PROGRAM Backbone
VAR
	RTC_FB					: RTC;
	NT_GetTime_FB			: NT_GetTime;
	RTCManagement_FB		: RTCManagement;
	FB_GetLocalAmsNetId_LU	: fb_GetLocalAmsNetId;
	bAborted				: BOOL;
	Blink_Abort				: BLINK;
	bError					: BOOL;
	Blink_Error				: BLINK;
	
	//Recipe Line 1
	Recipe_1				: FB_Recipe;
	CustomPattern_1			: RobotCustomPattern;
	Layer_1					: FB_Layer;
	
	//Recipe Line 2
	Recipe_2				: FB_Recipe;
	CustomPattern_2			: RobotCustomPattern;
	Layer_2					: FB_Layer;
	
	//Recipe Line 3
	Recipe_3				: FB_Recipe;
	CustomPattern_3			: RobotCustomPattern;
	Layer_3					: FB_Layer;
	
	//Recipe Line 4
	Recipe_4				: FB_Recipe;
	CustomPattern_4			: RobotCustomPattern;
	Layer_4					: FB_Layer;
	
	//Data Collect
	DataCollect_Palletizing_1: FGHS_DataCollect_Palletizing;
	DataCollect_Palletizing_2: FGHS_DataCollect_Palletizing;
	DataCollect_Palletizing_3: FGHS_DataCollect_Palletizing;
	DataCollect_Palletizing_4: FGHS_DataCollect_Palletizing;
	
	CheckCounter			: ARRAY [1..4] OF USINT;
	Index					: ARRAY [1..4] OF INT;
	RotatePicking			: RotatePick;
	AlarmEventHistory		: ARRAY[1..100] OF Alarm_Event_History;
	AlarmEventActive		: ARRAY[1..100] OF Alarm_Event_Active;
	OEE_Time				: OEETime;
	OEE_Time_Outfeed		: OEETime;
	bWarning				: BOOL;
	Blink_Warning			: BLINK;
	TON_Full				: TON;
	bRequest				: BOOL;
	bReleased				: BOOL;
	CheckShuttle			: FB_CheckShuttlePos;
	Check_Door				: TON;
	String_Time				: STRING(255);
	OEE_Counter				: ARRAY [1..4] OF OEECounter;
END_VAR
VAR // added by the converter: edge detectors and wires of the graphical bodies
    _w1 : BOOL;
    _rt1 : R_TRIG;
END_VAR

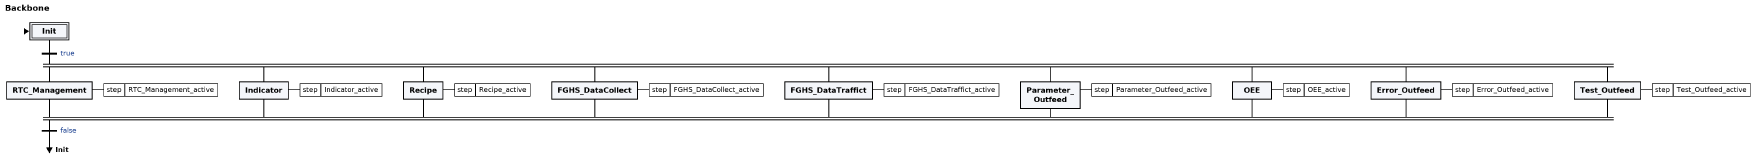
INITIAL_STEP Init:
END_STEP
TRANSITION FROM Init TO (RTC_Management, Indicator, Recipe, FGHS_DataCollect, FGHS_DataTraffict, Parameter_Outfeed, OEE, Error_Outfeed, Test_Outfeed)
    := true;
END_TRANSITION
STEP RTC_Management:
    RTC_Management_active(N);  // step action
END_STEP
STEP Indicator:
    Indicator_active(N);  // step action
END_STEP
STEP Recipe:
    Recipe_active(N);  // step action
END_STEP
STEP FGHS_DataCollect:
    FGHS_DataCollect_active(N);  // step action
END_STEP
STEP FGHS_DataTraffict:
    FGHS_DataTraffict_active(N);  // step action
END_STEP
STEP Parameter_Outfeed:
    Parameter_Outfeed_active(N);  // step action
END_STEP
STEP OEE:
    OEE_active(N);  // step action
END_STEP
STEP Error_Outfeed:
    Error_Outfeed_active(N);  // step action
END_STEP
STEP Test_Outfeed:
    Test_Outfeed_active(N);  // step action
END_STEP
TRANSITION FROM (RTC_Management, Indicator, Recipe, FGHS_DataCollect, FGHS_DataTraffict, Parameter_Outfeed, OEE, Error_Outfeed, Test_Outfeed) TO Init
    := false;
END_TRANSITION

ACTION Error_Outfeed_active:
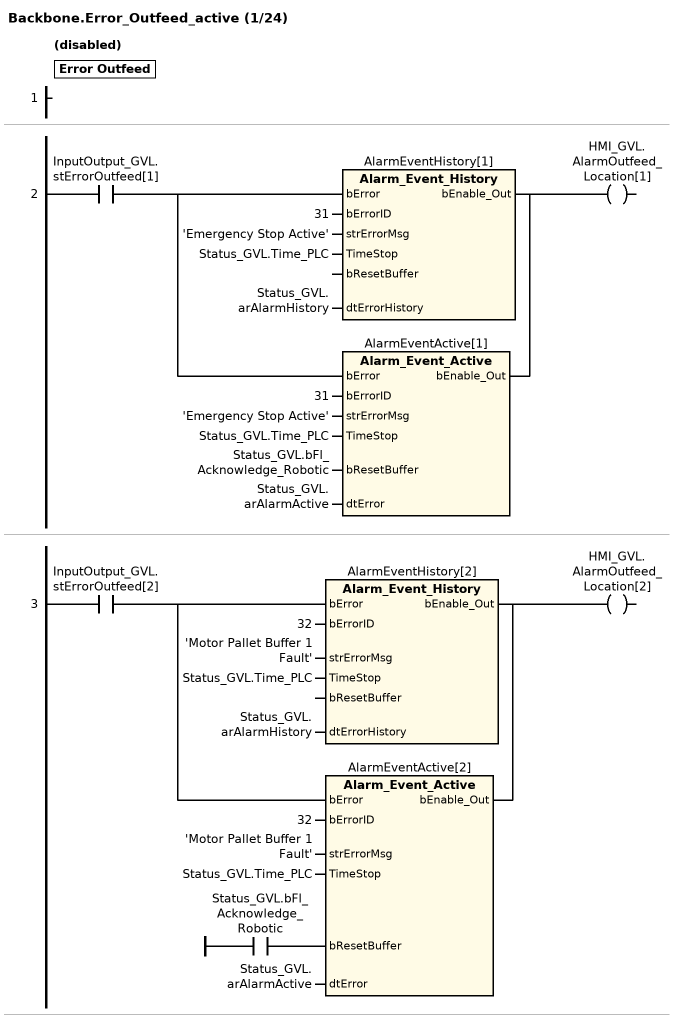
// NETWORK 1 (disabled)
// label: Error Outfeed

// NETWORK 2
AlarmEventHistory[1](
    bError := InputOutput_GVL.stErrorOutfeed[1],
    bErrorID := 31,
    strErrorMsg := 'Emergency Stop Active',
    TimeStop := Status_GVL.Time_PLC,
    dtErrorHistory := Status_GVL.arAlarmHistory); // Alarm_Event_History
AlarmEventActive[1](
    bError := InputOutput_GVL.stErrorOutfeed[1],
    bErrorID := 31,
    strErrorMsg := 'Emergency Stop Active',
    TimeStop := Status_GVL.Time_PLC,
    bResetBuffer := Status_GVL.bFl_Acknowledge_Robotic,
    dtError := Status_GVL.arAlarmActive); // Alarm_Event_Active
HMI_GVL.AlarmOutfeed_Location[1] := AlarmEventHistory[1].bEnable_Out OR AlarmEventActive[1].bEnable_Out;

// NETWORK 3
AlarmEventHistory[2](
    bError := InputOutput_GVL.stErrorOutfeed[2],
    bErrorID := 32,
    strErrorMsg := 'Motor Pallet Buffer 1 Fault',
    TimeStop := Status_GVL.Time_PLC,
    dtErrorHistory := Status_GVL.arAlarmHistory); // Alarm_Event_History
AlarmEventActive[2](
    bError := InputOutput_GVL.stErrorOutfeed[2],
    bErrorID := 32,
    strErrorMsg := 'Motor Pallet Buffer 1 Fault',
    TimeStop := Status_GVL.Time_PLC,
    bResetBuffer := Status_GVL.bFl_Acknowledge_Robotic,
    dtError := Status_GVL.arAlarmActive); // Alarm_Event_Active
HMI_GVL.AlarmOutfeed_Location[2] := AlarmEventHistory[2].bEnable_Out OR AlarmEventActive[2].bEnable_Out;

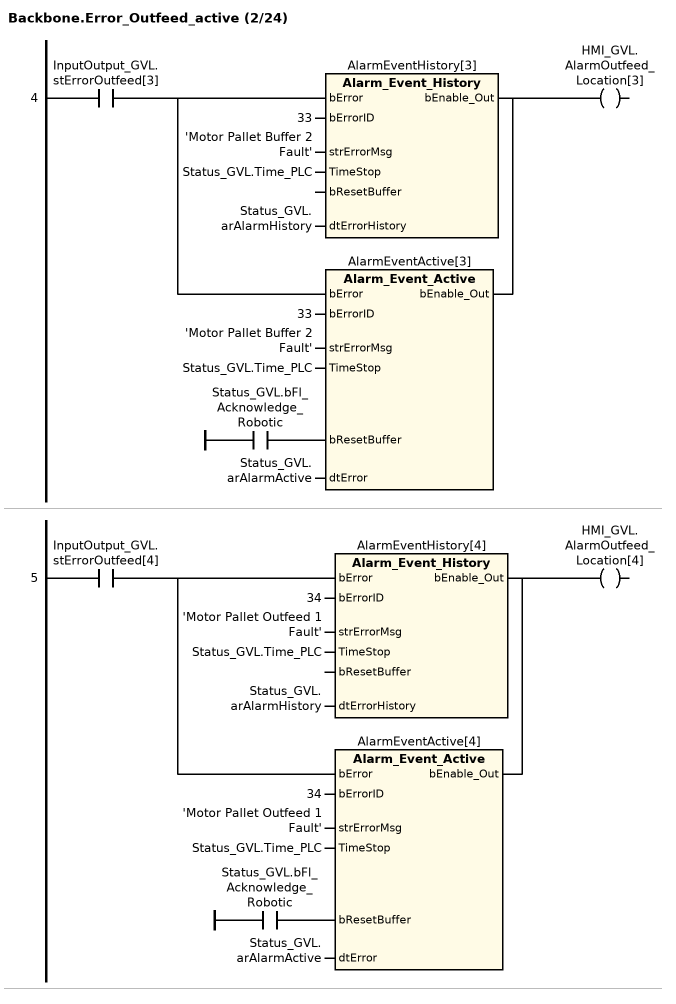
// NETWORK 4
AlarmEventHistory[3](
    bError := InputOutput_GVL.stErrorOutfeed[3],
    bErrorID := 33,
    strErrorMsg := 'Motor Pallet Buffer 2 Fault',
    TimeStop := Status_GVL.Time_PLC,
    dtErrorHistory := Status_GVL.arAlarmHistory); // Alarm_Event_History
AlarmEventActive[3](
    bError := InputOutput_GVL.stErrorOutfeed[3],
    bErrorID := 33,
    strErrorMsg := 'Motor Pallet Buffer 2 Fault',
    TimeStop := Status_GVL.Time_PLC,
    bResetBuffer := Status_GVL.bFl_Acknowledge_Robotic,
    dtError := Status_GVL.arAlarmActive); // Alarm_Event_Active
HMI_GVL.AlarmOutfeed_Location[3] := AlarmEventHistory[3].bEnable_Out OR AlarmEventActive[3].bEnable_Out;

// NETWORK 5
AlarmEventHistory[4](
    bError := InputOutput_GVL.stErrorOutfeed[4],
    bErrorID := 34,
    strErrorMsg := 'Motor Pallet Outfeed 1 Fault',
    TimeStop := Status_GVL.Time_PLC,
    dtErrorHistory := Status_GVL.arAlarmHistory); // Alarm_Event_History
AlarmEventActive[4](
    bError := InputOutput_GVL.stErrorOutfeed[4],
    bErrorID := 34,
    strErrorMsg := 'Motor Pallet Outfeed 1 Fault',
    TimeStop := Status_GVL.Time_PLC,
    bResetBuffer := Status_GVL.bFl_Acknowledge_Robotic,
    dtError := Status_GVL.arAlarmActive); // Alarm_Event_Active
HMI_GVL.AlarmOutfeed_Location[4] := AlarmEventHistory[4].bEnable_Out OR AlarmEventActive[4].bEnable_Out;

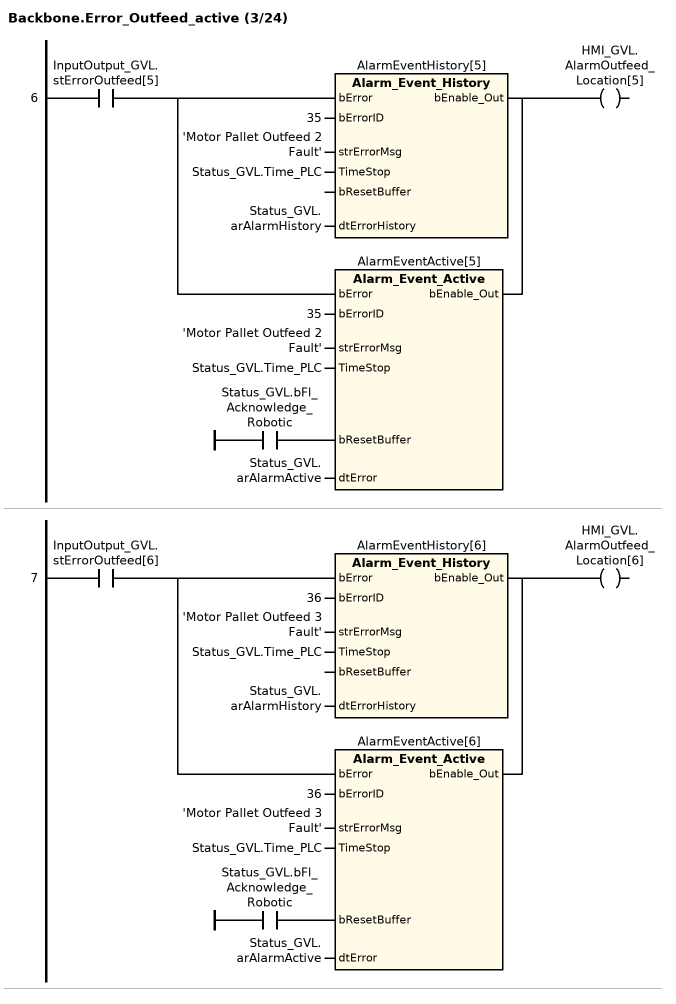
// NETWORK 6
AlarmEventHistory[5](
    bError := InputOutput_GVL.stErrorOutfeed[5],
    bErrorID := 35,
    strErrorMsg := 'Motor Pallet Outfeed 2 Fault',
    TimeStop := Status_GVL.Time_PLC,
    dtErrorHistory := Status_GVL.arAlarmHistory); // Alarm_Event_History
AlarmEventActive[5](
    bError := InputOutput_GVL.stErrorOutfeed[5],
    bErrorID := 35,
    strErrorMsg := 'Motor Pallet Outfeed 2 Fault',
    TimeStop := Status_GVL.Time_PLC,
    bResetBuffer := Status_GVL.bFl_Acknowledge_Robotic,
    dtError := Status_GVL.arAlarmActive); // Alarm_Event_Active
HMI_GVL.AlarmOutfeed_Location[5] := AlarmEventHistory[5].bEnable_Out OR AlarmEventActive[5].bEnable_Out;

// NETWORK 7
AlarmEventHistory[6](
    bError := InputOutput_GVL.stErrorOutfeed[6],
    bErrorID := 36,
    strErrorMsg := 'Motor Pallet Outfeed 3 Fault',
    TimeStop := Status_GVL.Time_PLC,
    dtErrorHistory := Status_GVL.arAlarmHistory); // Alarm_Event_History
AlarmEventActive[6](
    bError := InputOutput_GVL.stErrorOutfeed[6],
    bErrorID := 36,
    strErrorMsg := 'Motor Pallet Outfeed 3 Fault',
    TimeStop := Status_GVL.Time_PLC,
    bResetBuffer := Status_GVL.bFl_Acknowledge_Robotic,
    dtError := Status_GVL.arAlarmActive); // Alarm_Event_Active
HMI_GVL.AlarmOutfeed_Location[6] := AlarmEventHistory[6].bEnable_Out OR AlarmEventActive[6].bEnable_Out;

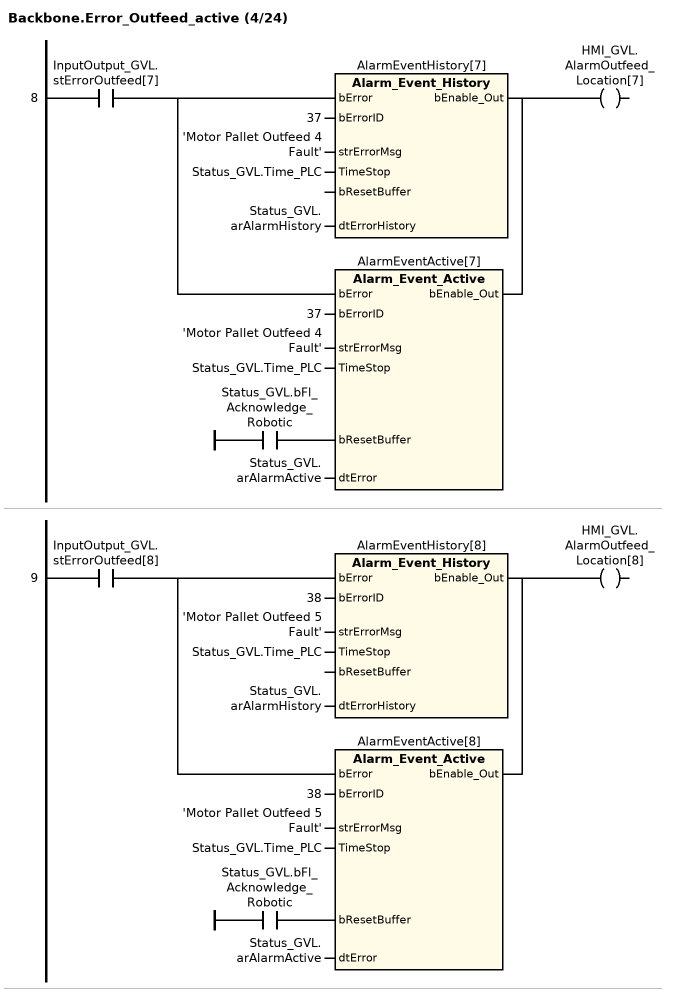
// NETWORK 8
AlarmEventHistory[7](
    bError := InputOutput_GVL.stErrorOutfeed[7],
    bErrorID := 37,
    strErrorMsg := 'Motor Pallet Outfeed 4 Fault',
    TimeStop := Status_GVL.Time_PLC,
    dtErrorHistory := Status_GVL.arAlarmHistory); // Alarm_Event_History
AlarmEventActive[7](
    bError := InputOutput_GVL.stErrorOutfeed[7],
    bErrorID := 37,
    strErrorMsg := 'Motor Pallet Outfeed 4 Fault',
    TimeStop := Status_GVL.Time_PLC,
    bResetBuffer := Status_GVL.bFl_Acknowledge_Robotic,
    dtError := Status_GVL.arAlarmActive); // Alarm_Event_Active
HMI_GVL.AlarmOutfeed_Location[7] := AlarmEventHistory[7].bEnable_Out OR AlarmEventActive[7].bEnable_Out;

// NETWORK 9
AlarmEventHistory[8](
    bError := InputOutput_GVL.stErrorOutfeed[8],
    bErrorID := 38,
    strErrorMsg := 'Motor Pallet Outfeed 5 Fault',
    TimeStop := Status_GVL.Time_PLC,
    dtErrorHistory := Status_GVL.arAlarmHistory); // Alarm_Event_History
AlarmEventActive[8](
    bError := InputOutput_GVL.stErrorOutfeed[8],
    bErrorID := 38,
    strErrorMsg := 'Motor Pallet Outfeed 5 Fault',
    TimeStop := Status_GVL.Time_PLC,
    bResetBuffer := Status_GVL.bFl_Acknowledge_Robotic,
    dtError := Status_GVL.arAlarmActive); // Alarm_Event_Active
HMI_GVL.AlarmOutfeed_Location[8] := AlarmEventHistory[8].bEnable_Out OR AlarmEventActive[8].bEnable_Out;

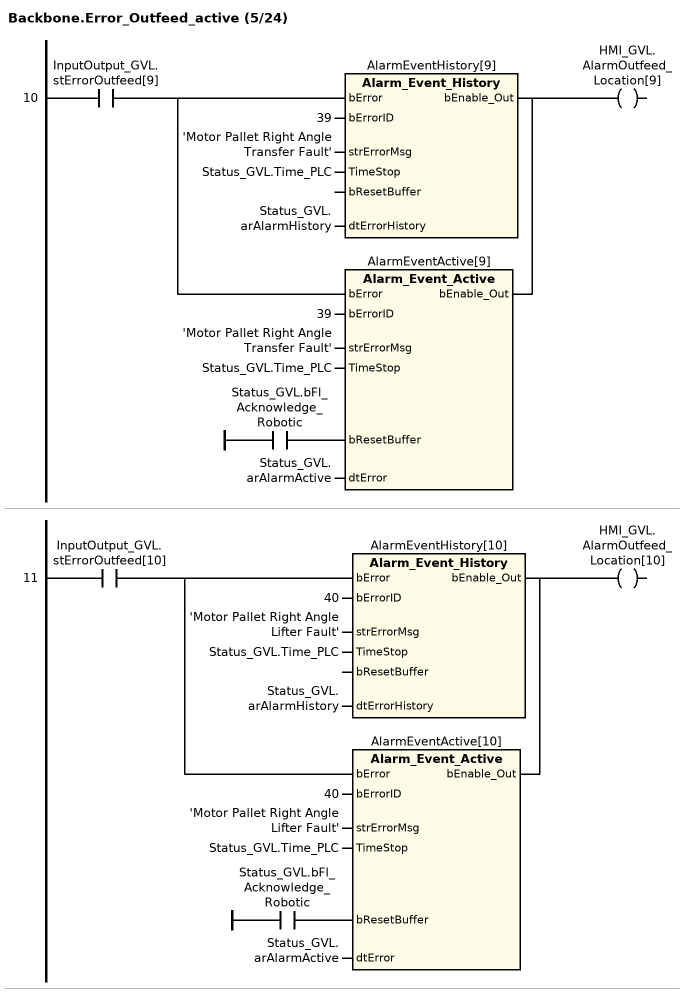
// NETWORK 10
AlarmEventHistory[9](
    bError := InputOutput_GVL.stErrorOutfeed[9],
    bErrorID := 39,
    strErrorMsg := 'Motor Pallet Right Angle Transfer Fault',
    TimeStop := Status_GVL.Time_PLC,
    dtErrorHistory := Status_GVL.arAlarmHistory); // Alarm_Event_History
AlarmEventActive[9](
    bError := InputOutput_GVL.stErrorOutfeed[9],
    bErrorID := 39,
    strErrorMsg := 'Motor Pallet Right Angle Transfer Fault',
    TimeStop := Status_GVL.Time_PLC,
    bResetBuffer := Status_GVL.bFl_Acknowledge_Robotic,
    dtError := Status_GVL.arAlarmActive); // Alarm_Event_Active
HMI_GVL.AlarmOutfeed_Location[9] := AlarmEventHistory[9].bEnable_Out OR AlarmEventActive[9].bEnable_Out;

// NETWORK 11
AlarmEventHistory[10](
    bError := InputOutput_GVL.stErrorOutfeed[10],
    bErrorID := 40,
    strErrorMsg := 'Motor Pallet Right Angle Lifter Fault',
    TimeStop := Status_GVL.Time_PLC,
    dtErrorHistory := Status_GVL.arAlarmHistory); // Alarm_Event_History
AlarmEventActive[10](
    bError := InputOutput_GVL.stErrorOutfeed[10],
    bErrorID := 40,
    strErrorMsg := 'Motor Pallet Right Angle Lifter Fault',
    TimeStop := Status_GVL.Time_PLC,
    bResetBuffer := Status_GVL.bFl_Acknowledge_Robotic,
    dtError := Status_GVL.arAlarmActive); // Alarm_Event_Active
HMI_GVL.AlarmOutfeed_Location[10] := AlarmEventHistory[10].bEnable_Out OR AlarmEventActive[10].bEnable_Out;

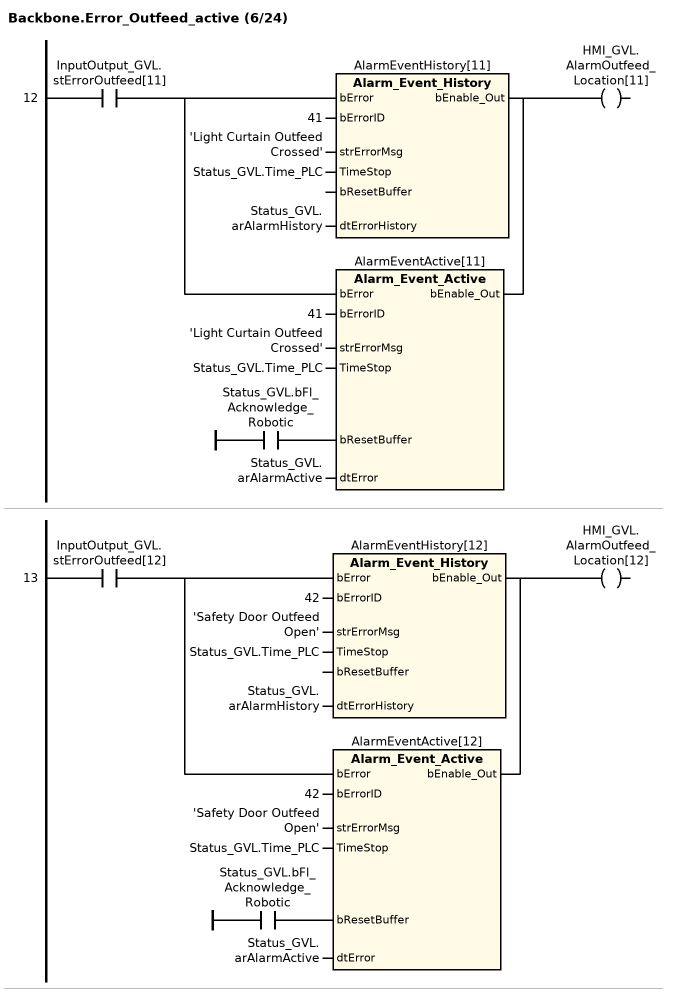
// NETWORK 12
AlarmEventHistory[11](
    bError := InputOutput_GVL.stErrorOutfeed[11],
    bErrorID := 41,
    strErrorMsg := 'Light Curtain Outfeed Crossed',
    TimeStop := Status_GVL.Time_PLC,
    dtErrorHistory := Status_GVL.arAlarmHistory); // Alarm_Event_History
AlarmEventActive[11](
    bError := InputOutput_GVL.stErrorOutfeed[11],
    bErrorID := 41,
    strErrorMsg := 'Light Curtain Outfeed Crossed',
    TimeStop := Status_GVL.Time_PLC,
    bResetBuffer := Status_GVL.bFl_Acknowledge_Robotic,
    dtError := Status_GVL.arAlarmActive); // Alarm_Event_Active
HMI_GVL.AlarmOutfeed_Location[11] := AlarmEventHistory[11].bEnable_Out OR AlarmEventActive[11].bEnable_Out;

// NETWORK 13
AlarmEventHistory[12](
    bError := InputOutput_GVL.stErrorOutfeed[12],
    bErrorID := 42,
    strErrorMsg := 'Safety Door Outfeed Open',
    TimeStop := Status_GVL.Time_PLC,
    dtErrorHistory := Status_GVL.arAlarmHistory); // Alarm_Event_History
AlarmEventActive[12](
    bError := InputOutput_GVL.stErrorOutfeed[12],
    bErrorID := 42,
    strErrorMsg := 'Safety Door Outfeed Open',
    TimeStop := Status_GVL.Time_PLC,
    bResetBuffer := Status_GVL.bFl_Acknowledge_Robotic,
    dtError := Status_GVL.arAlarmActive); // Alarm_Event_Active
HMI_GVL.AlarmOutfeed_Location[12] := AlarmEventHistory[12].bEnable_Out OR AlarmEventActive[12].bEnable_Out;

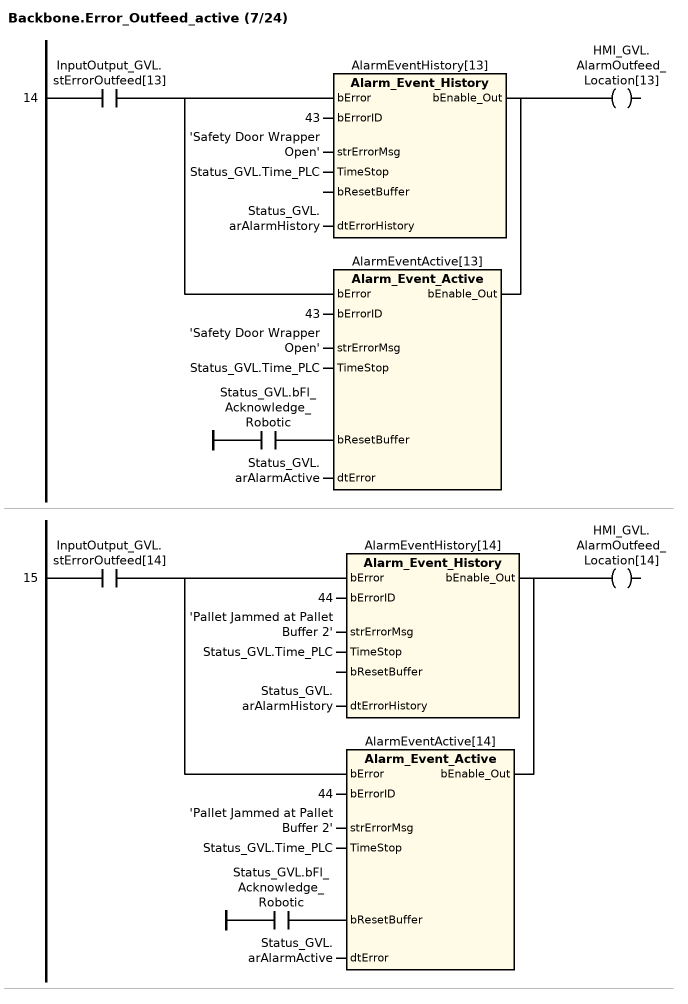
// NETWORK 14
AlarmEventHistory[13](
    bError := InputOutput_GVL.stErrorOutfeed[13],
    bErrorID := 43,
    strErrorMsg := 'Safety Door Wrapper Open',
    TimeStop := Status_GVL.Time_PLC,
    dtErrorHistory := Status_GVL.arAlarmHistory); // Alarm_Event_History
AlarmEventActive[13](
    bError := InputOutput_GVL.stErrorOutfeed[13],
    bErrorID := 43,
    strErrorMsg := 'Safety Door Wrapper Open',
    TimeStop := Status_GVL.Time_PLC,
    bResetBuffer := Status_GVL.bFl_Acknowledge_Robotic,
    dtError := Status_GVL.arAlarmActive); // Alarm_Event_Active
HMI_GVL.AlarmOutfeed_Location[13] := AlarmEventHistory[13].bEnable_Out OR AlarmEventActive[13].bEnable_Out;

// NETWORK 15
AlarmEventHistory[14](
    bError := InputOutput_GVL.stErrorOutfeed[14],
    bErrorID := 44,
    strErrorMsg := 'Pallet Jammed at Pallet Buffer 2',
    TimeStop := Status_GVL.Time_PLC,
    dtErrorHistory := Status_GVL.arAlarmHistory); // Alarm_Event_History
AlarmEventActive[14](
    bError := InputOutput_GVL.stErrorOutfeed[14],
    bErrorID := 44,
    strErrorMsg := 'Pallet Jammed at Pallet Buffer 2',
    TimeStop := Status_GVL.Time_PLC,
    bResetBuffer := Status_GVL.bFl_Acknowledge_Robotic,
    dtError := Status_GVL.arAlarmActive); // Alarm_Event_Active
HMI_GVL.AlarmOutfeed_Location[14] := AlarmEventHistory[14].bEnable_Out OR AlarmEventActive[14].bEnable_Out;

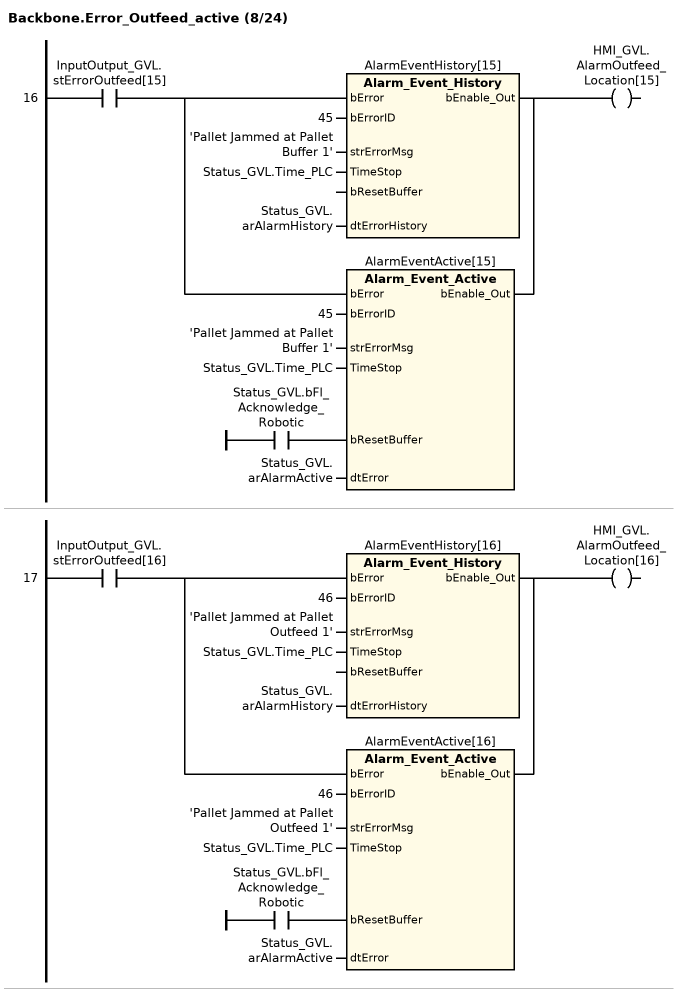
// NETWORK 16
AlarmEventHistory[15](
    bError := InputOutput_GVL.stErrorOutfeed[15],
    bErrorID := 45,
    strErrorMsg := 'Pallet Jammed at Pallet Buffer 1',
    TimeStop := Status_GVL.Time_PLC,
    dtErrorHistory := Status_GVL.arAlarmHistory); // Alarm_Event_History
AlarmEventActive[15](
    bError := InputOutput_GVL.stErrorOutfeed[15],
    bErrorID := 45,
    strErrorMsg := 'Pallet Jammed at Pallet Buffer 1',
    TimeStop := Status_GVL.Time_PLC,
    bResetBuffer := Status_GVL.bFl_Acknowledge_Robotic,
    dtError := Status_GVL.arAlarmActive); // Alarm_Event_Active
HMI_GVL.AlarmOutfeed_Location[15] := AlarmEventHistory[15].bEnable_Out OR AlarmEventActive[15].bEnable_Out;

// NETWORK 17
AlarmEventHistory[16](
    bError := InputOutput_GVL.stErrorOutfeed[16],
    bErrorID := 46,
    strErrorMsg := 'Pallet Jammed at Pallet Outfeed 1',
    TimeStop := Status_GVL.Time_PLC,
    dtErrorHistory := Status_GVL.arAlarmHistory); // Alarm_Event_History
AlarmEventActive[16](
    bError := InputOutput_GVL.stErrorOutfeed[16],
    bErrorID := 46,
    strErrorMsg := 'Pallet Jammed at Pallet Outfeed 1',
    TimeStop := Status_GVL.Time_PLC,
    bResetBuffer := Status_GVL.bFl_Acknowledge_Robotic,
    dtError := Status_GVL.arAlarmActive); // Alarm_Event_Active
HMI_GVL.AlarmOutfeed_Location[16] := AlarmEventHistory[16].bEnable_Out OR AlarmEventActive[16].bEnable_Out;

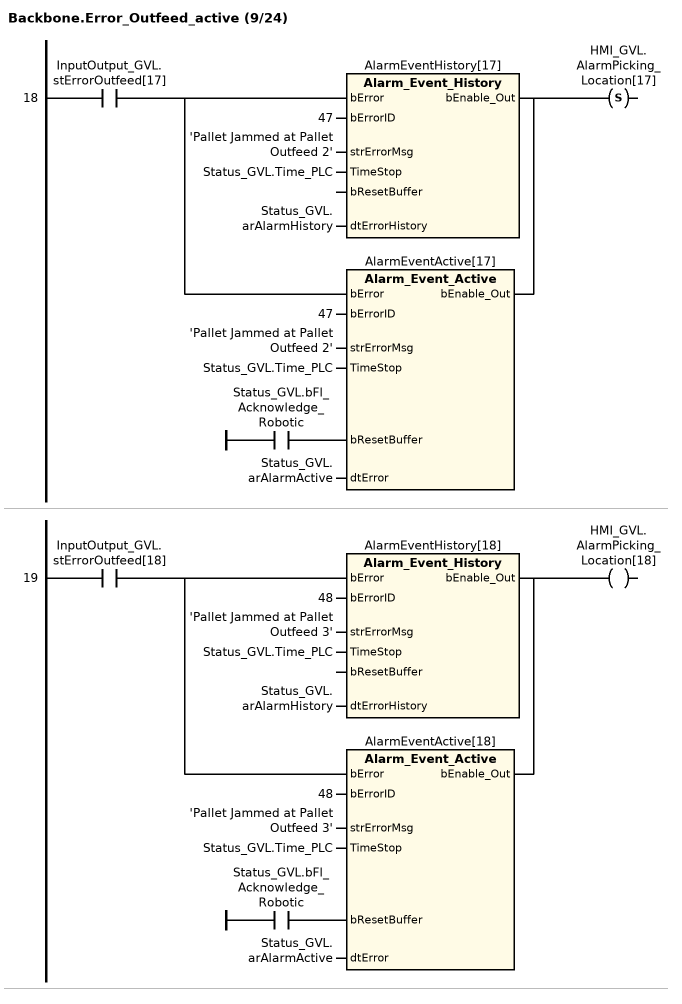
// NETWORK 18
AlarmEventHistory[17](
    bError := InputOutput_GVL.stErrorOutfeed[17],
    bErrorID := 47,
    strErrorMsg := 'Pallet Jammed at Pallet Outfeed 2',
    TimeStop := Status_GVL.Time_PLC,
    dtErrorHistory := Status_GVL.arAlarmHistory); // Alarm_Event_History
AlarmEventActive[17](
    bError := InputOutput_GVL.stErrorOutfeed[17],
    bErrorID := 47,
    strErrorMsg := 'Pallet Jammed at Pallet Outfeed 2',
    TimeStop := Status_GVL.Time_PLC,
    bResetBuffer := Status_GVL.bFl_Acknowledge_Robotic,
    dtError := Status_GVL.arAlarmActive); // Alarm_Event_Active
HMI_GVL.AlarmPicking_Location[17] S= AlarmEventHistory[17].bEnable_Out OR AlarmEventActive[17].bEnable_Out;

// NETWORK 19
AlarmEventHistory[18](
    bError := InputOutput_GVL.stErrorOutfeed[18],
    bErrorID := 48,
    strErrorMsg := 'Pallet Jammed at Pallet Outfeed 3',
    TimeStop := Status_GVL.Time_PLC,
    dtErrorHistory := Status_GVL.arAlarmHistory); // Alarm_Event_History
AlarmEventActive[18](
    bError := InputOutput_GVL.stErrorOutfeed[18],
    bErrorID := 48,
    strErrorMsg := 'Pallet Jammed at Pallet Outfeed 3',
    TimeStop := Status_GVL.Time_PLC,
    bResetBuffer := Status_GVL.bFl_Acknowledge_Robotic,
    dtError := Status_GVL.arAlarmActive); // Alarm_Event_Active
HMI_GVL.AlarmPicking_Location[18] := AlarmEventHistory[18].bEnable_Out OR AlarmEventActive[18].bEnable_Out;

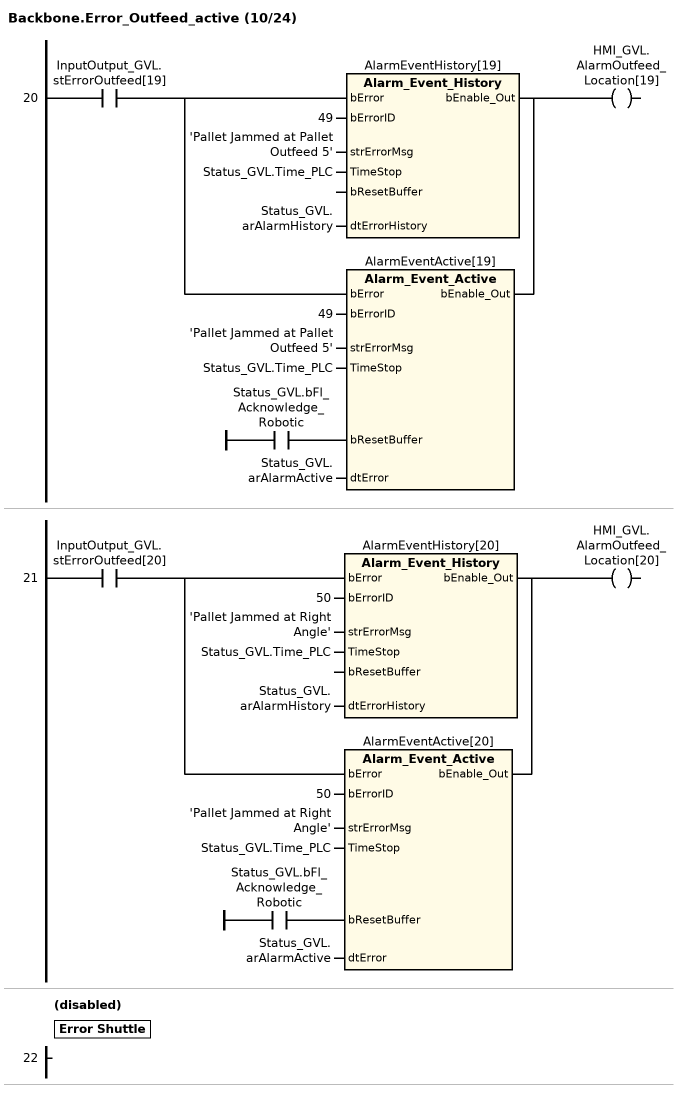
// NETWORK 20
AlarmEventHistory[19](
    bError := InputOutput_GVL.stErrorOutfeed[19],
    bErrorID := 49,
    strErrorMsg := 'Pallet Jammed at Pallet Outfeed 5',
    TimeStop := Status_GVL.Time_PLC,
    dtErrorHistory := Status_GVL.arAlarmHistory); // Alarm_Event_History
AlarmEventActive[19](
    bError := InputOutput_GVL.stErrorOutfeed[19],
    bErrorID := 49,
    strErrorMsg := 'Pallet Jammed at Pallet Outfeed 5',
    TimeStop := Status_GVL.Time_PLC,
    bResetBuffer := Status_GVL.bFl_Acknowledge_Robotic,
    dtError := Status_GVL.arAlarmActive); // Alarm_Event_Active
HMI_GVL.AlarmOutfeed_Location[19] := AlarmEventHistory[19].bEnable_Out OR AlarmEventActive[19].bEnable_Out;

// NETWORK 21
AlarmEventHistory[20](
    bError := InputOutput_GVL.stErrorOutfeed[20],
    bErrorID := 50,
    strErrorMsg := 'Pallet Jammed at Right Angle',
    TimeStop := Status_GVL.Time_PLC,
    dtErrorHistory := Status_GVL.arAlarmHistory); // Alarm_Event_History
AlarmEventActive[20](
    bError := InputOutput_GVL.stErrorOutfeed[20],
    bErrorID := 50,
    strErrorMsg := 'Pallet Jammed at Right Angle',
    TimeStop := Status_GVL.Time_PLC,
    bResetBuffer := Status_GVL.bFl_Acknowledge_Robotic,
    dtError := Status_GVL.arAlarmActive); // Alarm_Event_Active
HMI_GVL.AlarmOutfeed_Location[20] := AlarmEventHistory[20].bEnable_Out OR AlarmEventActive[20].bEnable_Out;

// NETWORK 22 (disabled)
// label: Error Shuttle

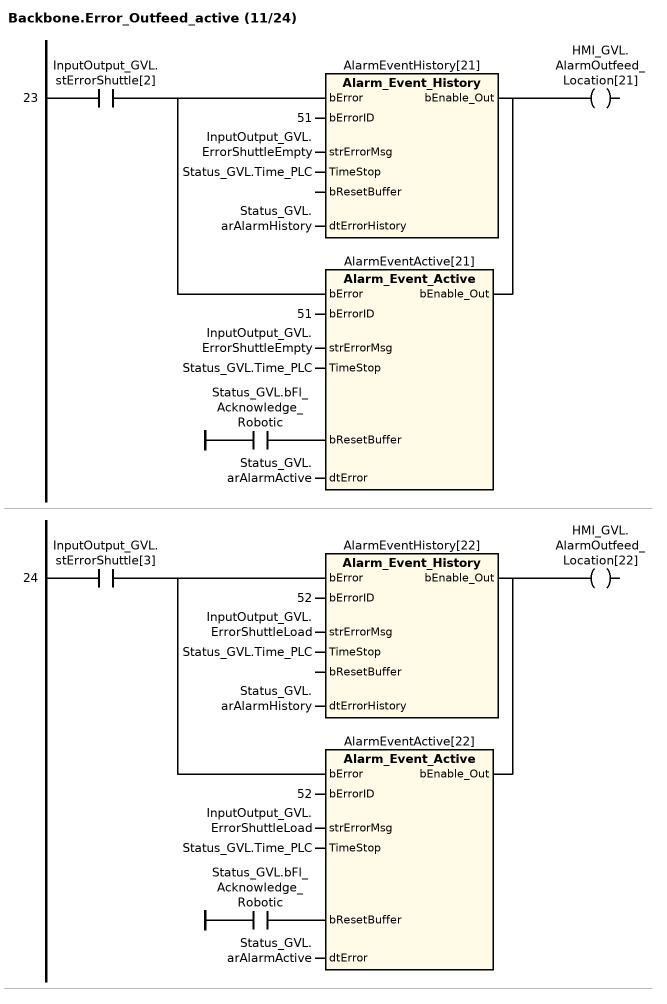
// NETWORK 23
AlarmEventHistory[21](
    bError := InputOutput_GVL.stErrorShuttle[2],
    bErrorID := 51,
    strErrorMsg := InputOutput_GVL.ErrorShuttleEmpty,
    TimeStop := Status_GVL.Time_PLC,
    dtErrorHistory := Status_GVL.arAlarmHistory); // Alarm_Event_History
AlarmEventActive[21](
    bError := InputOutput_GVL.stErrorShuttle[2],
    bErrorID := 51,
    strErrorMsg := InputOutput_GVL.ErrorShuttleEmpty,
    TimeStop := Status_GVL.Time_PLC,
    bResetBuffer := Status_GVL.bFl_Acknowledge_Robotic,
    dtError := Status_GVL.arAlarmActive); // Alarm_Event_Active
HMI_GVL.AlarmOutfeed_Location[21] := AlarmEventHistory[21].bEnable_Out OR AlarmEventActive[21].bEnable_Out;

// NETWORK 24
AlarmEventHistory[22](
    bError := InputOutput_GVL.stErrorShuttle[3],
    bErrorID := 52,
    strErrorMsg := InputOutput_GVL.ErrorShuttleLoad,
    TimeStop := Status_GVL.Time_PLC,
    dtErrorHistory := Status_GVL.arAlarmHistory); // Alarm_Event_History
AlarmEventActive[22](
    bError := InputOutput_GVL.stErrorShuttle[3],
    bErrorID := 52,
    strErrorMsg := InputOutput_GVL.ErrorShuttleLoad,
    TimeStop := Status_GVL.Time_PLC,
    bResetBuffer := Status_GVL.bFl_Acknowledge_Robotic,
    dtError := Status_GVL.arAlarmActive); // Alarm_Event_Active
HMI_GVL.AlarmOutfeed_Location[22] := AlarmEventHistory[22].bEnable_Out OR AlarmEventActive[22].bEnable_Out;

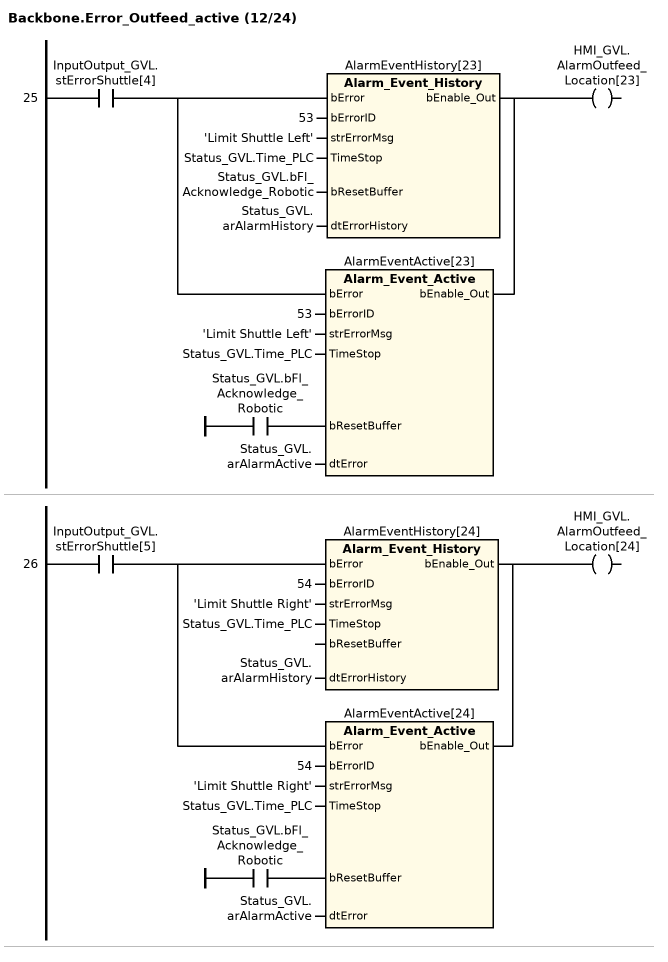
// NETWORK 25
AlarmEventHistory[23](
    bError := InputOutput_GVL.stErrorShuttle[4],
    bErrorID := 53,
    strErrorMsg := 'Limit Shuttle Left',
    TimeStop := Status_GVL.Time_PLC,
    bResetBuffer := Status_GVL.bFl_Acknowledge_Robotic,
    dtErrorHistory := Status_GVL.arAlarmHistory); // Alarm_Event_History
AlarmEventActive[23](
    bError := InputOutput_GVL.stErrorShuttle[4],
    bErrorID := 53,
    strErrorMsg := 'Limit Shuttle Left',
    TimeStop := Status_GVL.Time_PLC,
    bResetBuffer := Status_GVL.bFl_Acknowledge_Robotic,
    dtError := Status_GVL.arAlarmActive); // Alarm_Event_Active
HMI_GVL.AlarmOutfeed_Location[23] := AlarmEventHistory[23].bEnable_Out OR AlarmEventActive[23].bEnable_Out;

// NETWORK 26
AlarmEventHistory[24](
    bError := InputOutput_GVL.stErrorShuttle[5],
    bErrorID := 54,
    strErrorMsg := 'Limit Shuttle Right',
    TimeStop := Status_GVL.Time_PLC,
    dtErrorHistory := Status_GVL.arAlarmHistory); // Alarm_Event_History
AlarmEventActive[24](
    bError := InputOutput_GVL.stErrorShuttle[5],
    bErrorID := 54,
    strErrorMsg := 'Limit Shuttle Right',
    TimeStop := Status_GVL.Time_PLC,
    bResetBuffer := Status_GVL.bFl_Acknowledge_Robotic,
    dtError := Status_GVL.arAlarmActive); // Alarm_Event_Active
HMI_GVL.AlarmOutfeed_Location[24] := AlarmEventHistory[24].bEnable_Out OR AlarmEventActive[24].bEnable_Out;

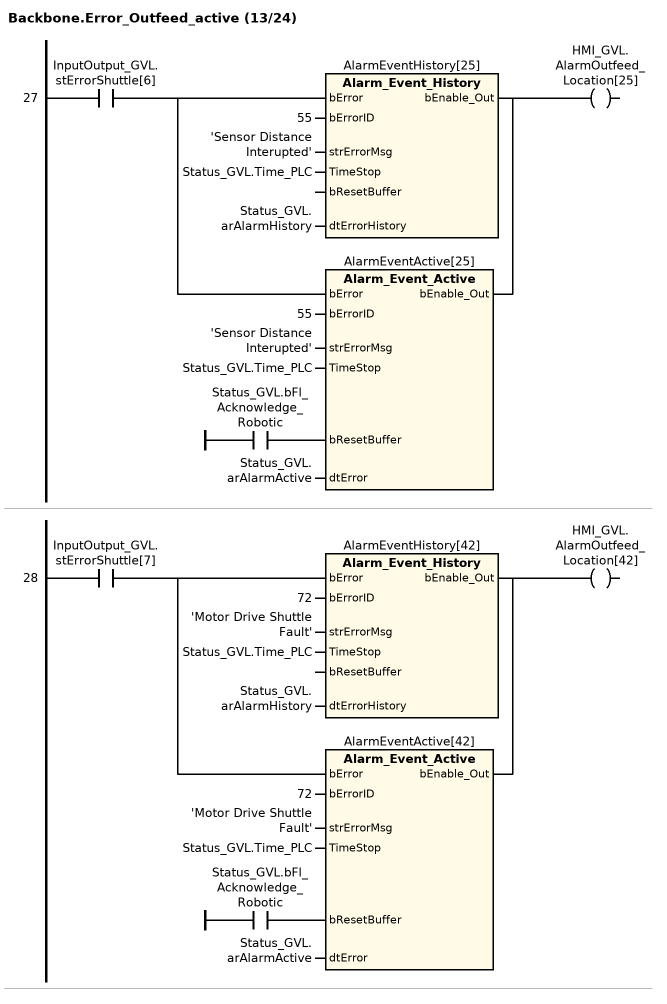
// NETWORK 27
AlarmEventHistory[25](
    bError := InputOutput_GVL.stErrorShuttle[6],
    bErrorID := 55,
    strErrorMsg := 'Sensor Distance Interupted',
    TimeStop := Status_GVL.Time_PLC,
    dtErrorHistory := Status_GVL.arAlarmHistory); // Alarm_Event_History
AlarmEventActive[25](
    bError := InputOutput_GVL.stErrorShuttle[6],
    bErrorID := 55,
    strErrorMsg := 'Sensor Distance Interupted',
    TimeStop := Status_GVL.Time_PLC,
    bResetBuffer := Status_GVL.bFl_Acknowledge_Robotic,
    dtError := Status_GVL.arAlarmActive); // Alarm_Event_Active
HMI_GVL.AlarmOutfeed_Location[25] := AlarmEventHistory[25].bEnable_Out OR AlarmEventActive[25].bEnable_Out;

// NETWORK 28
AlarmEventHistory[42](
    bError := InputOutput_GVL.stErrorShuttle[7],
    bErrorID := 72,
    strErrorMsg := 'Motor Drive Shuttle Fault',
    TimeStop := Status_GVL.Time_PLC,
    dtErrorHistory := Status_GVL.arAlarmHistory); // Alarm_Event_History
AlarmEventActive[42](
    bError := InputOutput_GVL.stErrorShuttle[7],
    bErrorID := 72,
    strErrorMsg := 'Motor Drive Shuttle Fault',
    TimeStop := Status_GVL.Time_PLC,
    bResetBuffer := Status_GVL.bFl_Acknowledge_Robotic,
    dtError := Status_GVL.arAlarmActive); // Alarm_Event_Active
HMI_GVL.AlarmOutfeed_Location[42] := AlarmEventHistory[42].bEnable_Out OR AlarmEventActive[42].bEnable_Out;

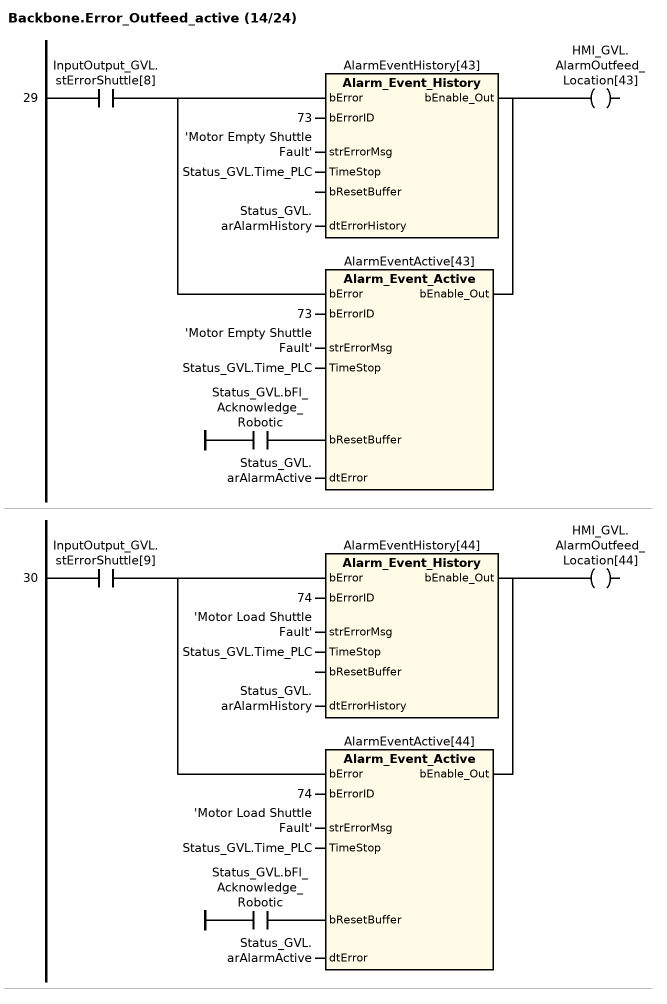
// NETWORK 29
AlarmEventHistory[43](
    bError := InputOutput_GVL.stErrorShuttle[8],
    bErrorID := 73,
    strErrorMsg := 'Motor Empty Shuttle Fault',
    TimeStop := Status_GVL.Time_PLC,
    dtErrorHistory := Status_GVL.arAlarmHistory); // Alarm_Event_History
AlarmEventActive[43](
    bError := InputOutput_GVL.stErrorShuttle[8],
    bErrorID := 73,
    strErrorMsg := 'Motor Empty Shuttle Fault',
    TimeStop := Status_GVL.Time_PLC,
    bResetBuffer := Status_GVL.bFl_Acknowledge_Robotic,
    dtError := Status_GVL.arAlarmActive); // Alarm_Event_Active
HMI_GVL.AlarmOutfeed_Location[43] := AlarmEventHistory[43].bEnable_Out OR AlarmEventActive[43].bEnable_Out;

// NETWORK 30
AlarmEventHistory[44](
    bError := InputOutput_GVL.stErrorShuttle[9],
    bErrorID := 74,
    strErrorMsg := 'Motor Load Shuttle Fault',
    TimeStop := Status_GVL.Time_PLC,
    dtErrorHistory := Status_GVL.arAlarmHistory); // Alarm_Event_History
AlarmEventActive[44](
    bError := InputOutput_GVL.stErrorShuttle[9],
    bErrorID := 74,
    strErrorMsg := 'Motor Load Shuttle Fault',
    TimeStop := Status_GVL.Time_PLC,
    bResetBuffer := Status_GVL.bFl_Acknowledge_Robotic,
    dtError := Status_GVL.arAlarmActive); // Alarm_Event_Active
HMI_GVL.AlarmOutfeed_Location[44] := AlarmEventHistory[44].bEnable_Out OR AlarmEventActive[44].bEnable_Out;

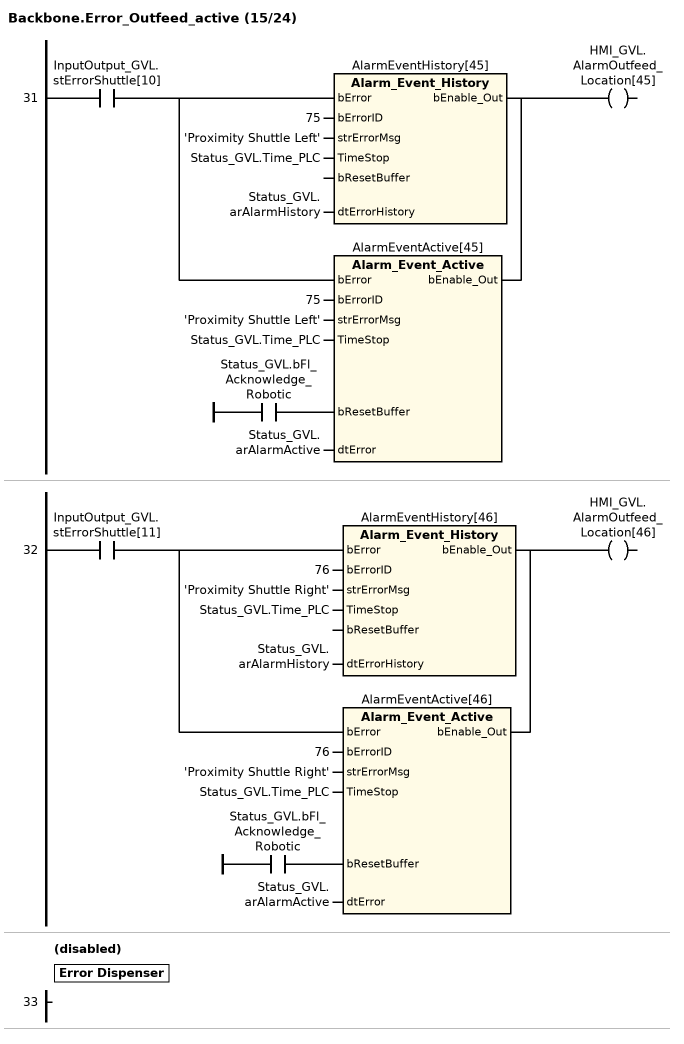
// NETWORK 31
AlarmEventHistory[45](
    bError := InputOutput_GVL.stErrorShuttle[10],
    bErrorID := 75,
    strErrorMsg := 'Proximity Shuttle Left',
    TimeStop := Status_GVL.Time_PLC,
    dtErrorHistory := Status_GVL.arAlarmHistory); // Alarm_Event_History
AlarmEventActive[45](
    bError := InputOutput_GVL.stErrorShuttle[10],
    bErrorID := 75,
    strErrorMsg := 'Proximity Shuttle Left',
    TimeStop := Status_GVL.Time_PLC,
    bResetBuffer := Status_GVL.bFl_Acknowledge_Robotic,
    dtError := Status_GVL.arAlarmActive); // Alarm_Event_Active
HMI_GVL.AlarmOutfeed_Location[45] := AlarmEventHistory[45].bEnable_Out OR AlarmEventActive[45].bEnable_Out;

// NETWORK 32
AlarmEventHistory[46](
    bError := InputOutput_GVL.stErrorShuttle[11],
    bErrorID := 76,
    strErrorMsg := 'Proximity Shuttle Right',
    TimeStop := Status_GVL.Time_PLC,
    dtErrorHistory := Status_GVL.arAlarmHistory); // Alarm_Event_History
AlarmEventActive[46](
    bError := InputOutput_GVL.stErrorShuttle[11],
    bErrorID := 76,
    strErrorMsg := 'Proximity Shuttle Right',
    TimeStop := Status_GVL.Time_PLC,
    bResetBuffer := Status_GVL.bFl_Acknowledge_Robotic,
    dtError := Status_GVL.arAlarmActive); // Alarm_Event_Active
HMI_GVL.AlarmOutfeed_Location[46] := AlarmEventHistory[46].bEnable_Out OR AlarmEventActive[46].bEnable_Out;

// NETWORK 33 (disabled)
// label: Error Dispenser

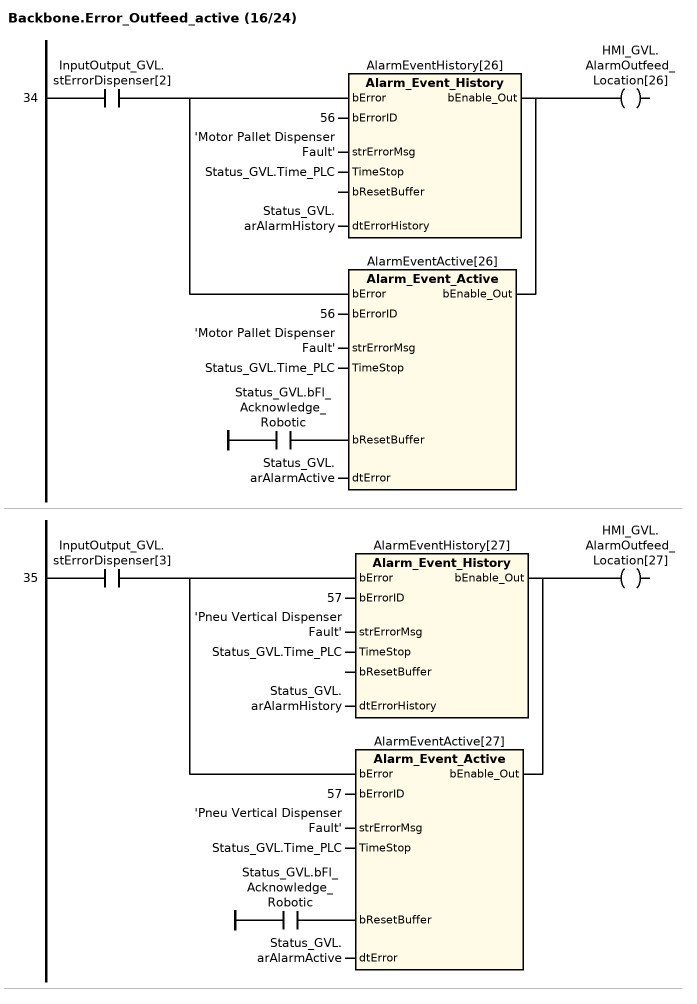
// NETWORK 34
AlarmEventHistory[26](
    bError := InputOutput_GVL.stErrorDispenser[2],
    bErrorID := 56,
    strErrorMsg := 'Motor Pallet Dispenser Fault',
    TimeStop := Status_GVL.Time_PLC,
    dtErrorHistory := Status_GVL.arAlarmHistory); // Alarm_Event_History
AlarmEventActive[26](
    bError := InputOutput_GVL.stErrorDispenser[2],
    bErrorID := 56,
    strErrorMsg := 'Motor Pallet Dispenser Fault',
    TimeStop := Status_GVL.Time_PLC,
    bResetBuffer := Status_GVL.bFl_Acknowledge_Robotic,
    dtError := Status_GVL.arAlarmActive); // Alarm_Event_Active
HMI_GVL.AlarmOutfeed_Location[26] := AlarmEventHistory[26].bEnable_Out OR AlarmEventActive[26].bEnable_Out;

// NETWORK 35
AlarmEventHistory[27](
    bError := InputOutput_GVL.stErrorDispenser[3],
    bErrorID := 57,
    strErrorMsg := 'Pneu Vertical Dispenser Fault',
    TimeStop := Status_GVL.Time_PLC,
    dtErrorHistory := Status_GVL.arAlarmHistory); // Alarm_Event_History
AlarmEventActive[27](
    bError := InputOutput_GVL.stErrorDispenser[3],
    bErrorID := 57,
    strErrorMsg := 'Pneu Vertical Dispenser Fault',
    TimeStop := Status_GVL.Time_PLC,
    bResetBuffer := Status_GVL.bFl_Acknowledge_Robotic,
    dtError := Status_GVL.arAlarmActive); // Alarm_Event_Active
HMI_GVL.AlarmOutfeed_Location[27] := AlarmEventHistory[27].bEnable_Out OR AlarmEventActive[27].bEnable_Out;

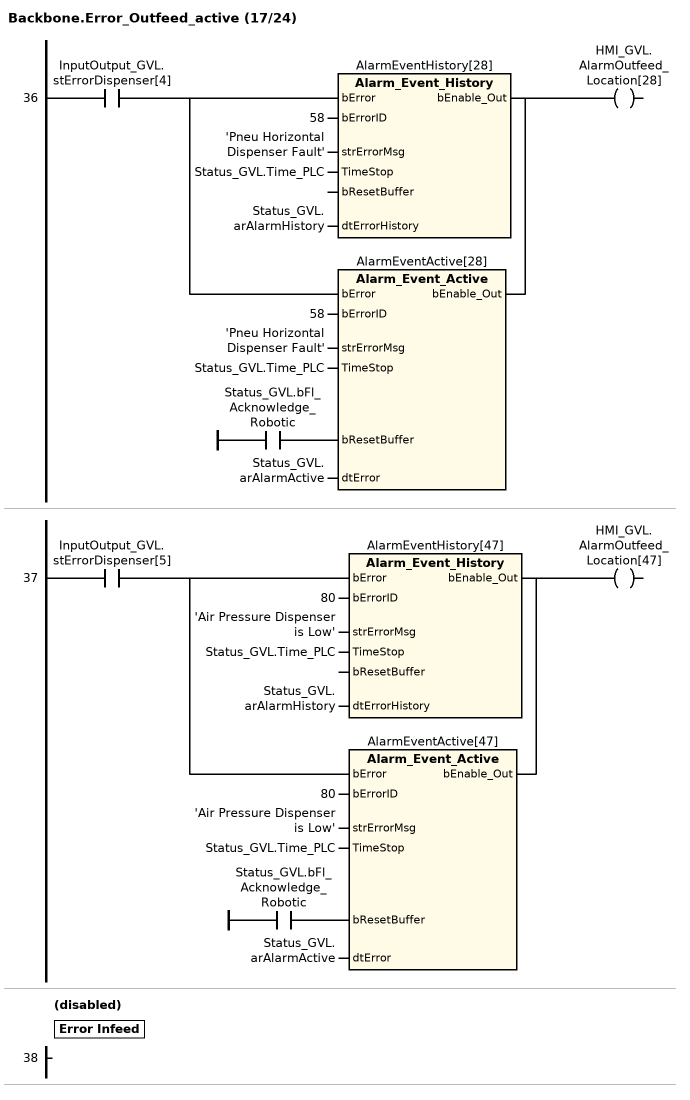
// NETWORK 36
AlarmEventHistory[28](
    bError := InputOutput_GVL.stErrorDispenser[4],
    bErrorID := 58,
    strErrorMsg := 'Pneu Horizontal Dispenser Fault',
    TimeStop := Status_GVL.Time_PLC,
    dtErrorHistory := Status_GVL.arAlarmHistory); // Alarm_Event_History
AlarmEventActive[28](
    bError := InputOutput_GVL.stErrorDispenser[4],
    bErrorID := 58,
    strErrorMsg := 'Pneu Horizontal Dispenser Fault',
    TimeStop := Status_GVL.Time_PLC,
    bResetBuffer := Status_GVL.bFl_Acknowledge_Robotic,
    dtError := Status_GVL.arAlarmActive); // Alarm_Event_Active
HMI_GVL.AlarmOutfeed_Location[28] := AlarmEventHistory[28].bEnable_Out OR AlarmEventActive[28].bEnable_Out;

// NETWORK 37
AlarmEventHistory[47](
    bError := InputOutput_GVL.stErrorDispenser[5],
    bErrorID := 80,
    strErrorMsg := 'Air Pressure Dispenser is Low',
    TimeStop := Status_GVL.Time_PLC,
    dtErrorHistory := Status_GVL.arAlarmHistory); // Alarm_Event_History
AlarmEventActive[47](
    bError := InputOutput_GVL.stErrorDispenser[5],
    bErrorID := 80,
    strErrorMsg := 'Air Pressure Dispenser is Low',
    TimeStop := Status_GVL.Time_PLC,
    bResetBuffer := Status_GVL.bFl_Acknowledge_Robotic,
    dtError := Status_GVL.arAlarmActive); // Alarm_Event_Active
HMI_GVL.AlarmOutfeed_Location[47] := AlarmEventHistory[47].bEnable_Out OR AlarmEventActive[47].bEnable_Out;

// NETWORK 38 (disabled)
// label: Error Infeed

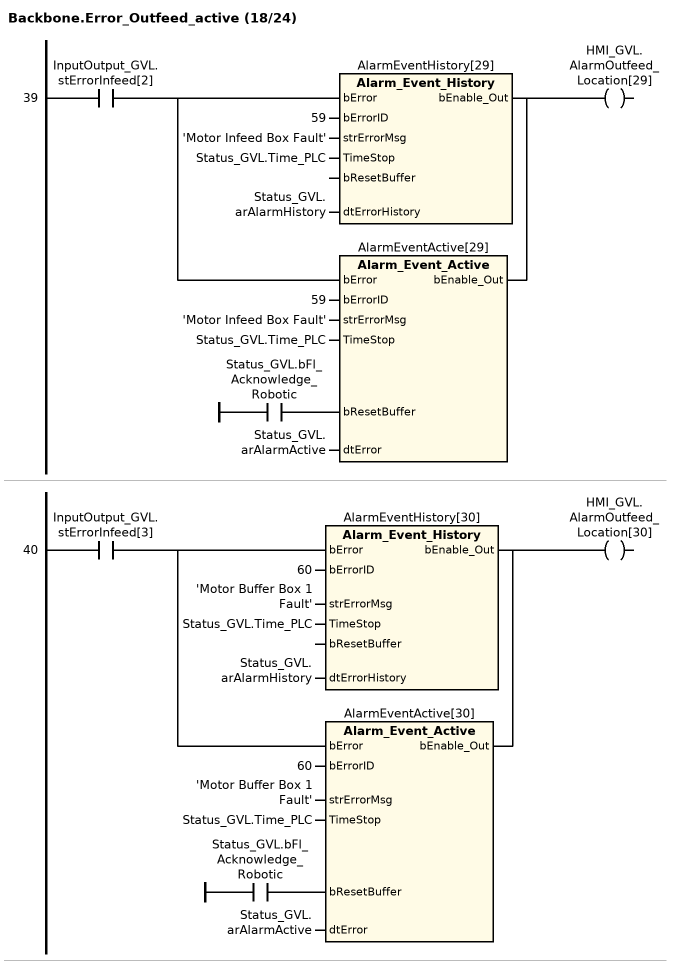
// NETWORK 39
AlarmEventHistory[29](
    bError := InputOutput_GVL.stErrorInfeed[2],
    bErrorID := 59,
    strErrorMsg := 'Motor Infeed Box Fault',
    TimeStop := Status_GVL.Time_PLC,
    dtErrorHistory := Status_GVL.arAlarmHistory); // Alarm_Event_History
AlarmEventActive[29](
    bError := InputOutput_GVL.stErrorInfeed[2],
    bErrorID := 59,
    strErrorMsg := 'Motor Infeed Box Fault',
    TimeStop := Status_GVL.Time_PLC,
    bResetBuffer := Status_GVL.bFl_Acknowledge_Robotic,
    dtError := Status_GVL.arAlarmActive); // Alarm_Event_Active
HMI_GVL.AlarmOutfeed_Location[29] := AlarmEventHistory[29].bEnable_Out OR AlarmEventActive[29].bEnable_Out;

// NETWORK 40
AlarmEventHistory[30](
    bError := InputOutput_GVL.stErrorInfeed[3],
    bErrorID := 60,
    strErrorMsg := 'Motor Buffer Box 1 Fault',
    TimeStop := Status_GVL.Time_PLC,
    dtErrorHistory := Status_GVL.arAlarmHistory); // Alarm_Event_History
AlarmEventActive[30](
    bError := InputOutput_GVL.stErrorInfeed[3],
    bErrorID := 60,
    strErrorMsg := 'Motor Buffer Box 1 Fault',
    TimeStop := Status_GVL.Time_PLC,
    bResetBuffer := Status_GVL.bFl_Acknowledge_Robotic,
    dtError := Status_GVL.arAlarmActive); // Alarm_Event_Active
HMI_GVL.AlarmOutfeed_Location[30] := AlarmEventHistory[30].bEnable_Out OR AlarmEventActive[30].bEnable_Out;

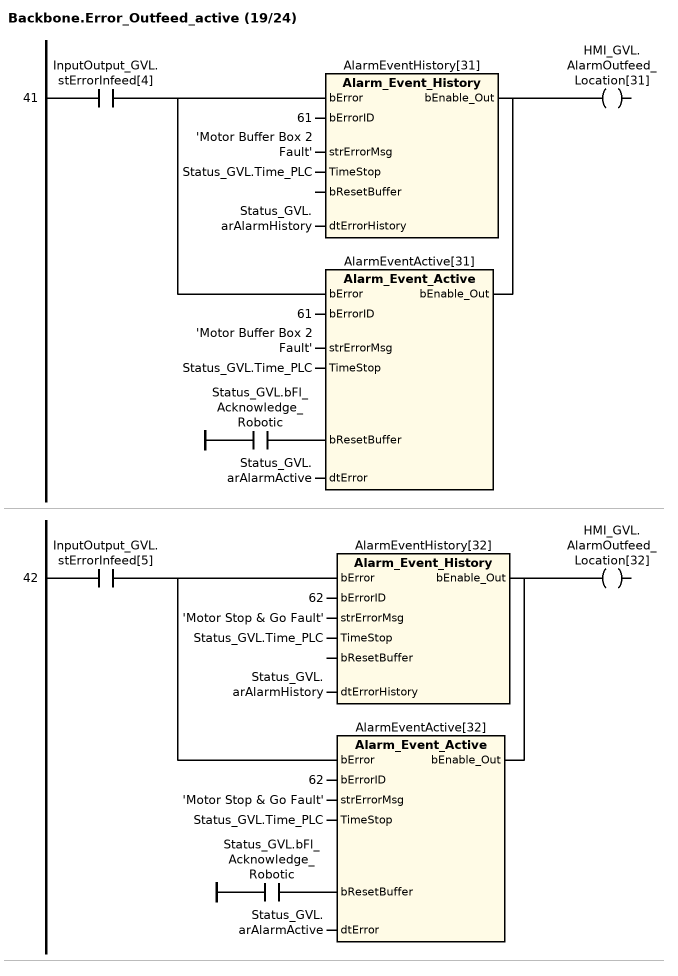
// NETWORK 41
AlarmEventHistory[31](
    bError := InputOutput_GVL.stErrorInfeed[4],
    bErrorID := 61,
    strErrorMsg := 'Motor Buffer Box 2 Fault',
    TimeStop := Status_GVL.Time_PLC,
    dtErrorHistory := Status_GVL.arAlarmHistory); // Alarm_Event_History
AlarmEventActive[31](
    bError := InputOutput_GVL.stErrorInfeed[4],
    bErrorID := 61,
    strErrorMsg := 'Motor Buffer Box 2 Fault',
    TimeStop := Status_GVL.Time_PLC,
    bResetBuffer := Status_GVL.bFl_Acknowledge_Robotic,
    dtError := Status_GVL.arAlarmActive); // Alarm_Event_Active
HMI_GVL.AlarmOutfeed_Location[31] := AlarmEventHistory[31].bEnable_Out OR AlarmEventActive[31].bEnable_Out;

// NETWORK 42
AlarmEventHistory[32](
    bError := InputOutput_GVL.stErrorInfeed[5],
    bErrorID := 62,
    strErrorMsg := 'Motor Stop & Go Fault',
    TimeStop := Status_GVL.Time_PLC,
    dtErrorHistory := Status_GVL.arAlarmHistory); // Alarm_Event_History
AlarmEventActive[32](
    bError := InputOutput_GVL.stErrorInfeed[5],
    bErrorID := 62,
    strErrorMsg := 'Motor Stop & Go Fault',
    TimeStop := Status_GVL.Time_PLC,
    bResetBuffer := Status_GVL.bFl_Acknowledge_Robotic,
    dtError := Status_GVL.arAlarmActive); // Alarm_Event_Active
HMI_GVL.AlarmOutfeed_Location[32] := AlarmEventHistory[32].bEnable_Out OR AlarmEventActive[32].bEnable_Out;

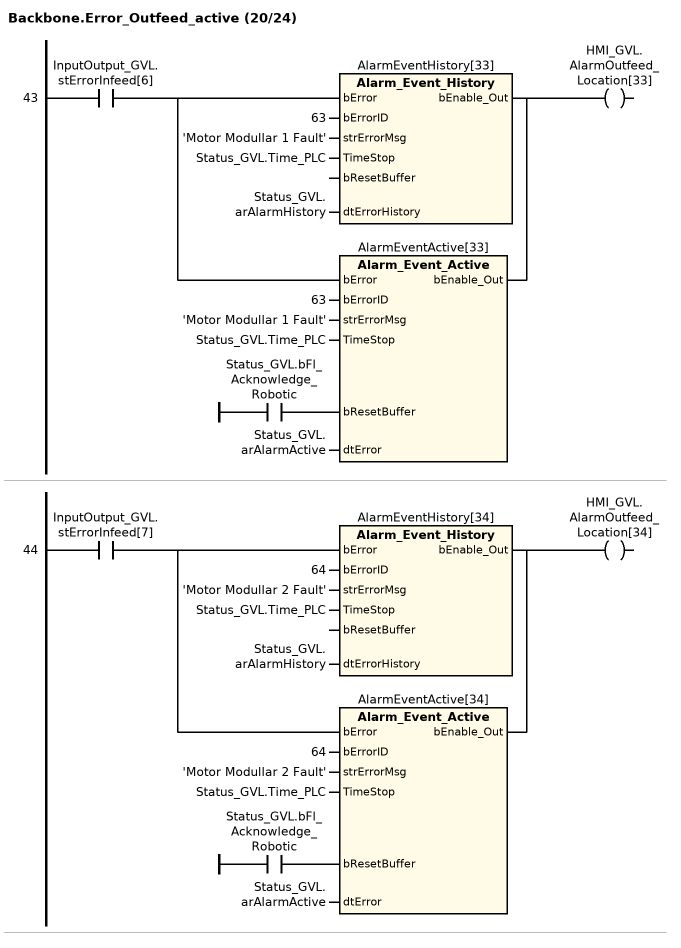
// NETWORK 43
AlarmEventHistory[33](
    bError := InputOutput_GVL.stErrorInfeed[6],
    bErrorID := 63,
    strErrorMsg := 'Motor Modullar 1 Fault',
    TimeStop := Status_GVL.Time_PLC,
    dtErrorHistory := Status_GVL.arAlarmHistory); // Alarm_Event_History
AlarmEventActive[33](
    bError := InputOutput_GVL.stErrorInfeed[6],
    bErrorID := 63,
    strErrorMsg := 'Motor Modullar 1 Fault',
    TimeStop := Status_GVL.Time_PLC,
    bResetBuffer := Status_GVL.bFl_Acknowledge_Robotic,
    dtError := Status_GVL.arAlarmActive); // Alarm_Event_Active
HMI_GVL.AlarmOutfeed_Location[33] := AlarmEventHistory[33].bEnable_Out OR AlarmEventActive[33].bEnable_Out;

// NETWORK 44
AlarmEventHistory[34](
    bError := InputOutput_GVL.stErrorInfeed[7],
    bErrorID := 64,
    strErrorMsg := 'Motor Modullar 2 Fault',
    TimeStop := Status_GVL.Time_PLC,
    dtErrorHistory := Status_GVL.arAlarmHistory); // Alarm_Event_History
AlarmEventActive[34](
    bError := InputOutput_GVL.stErrorInfeed[7],
    bErrorID := 64,
    strErrorMsg := 'Motor Modullar 2 Fault',
    TimeStop := Status_GVL.Time_PLC,
    bResetBuffer := Status_GVL.bFl_Acknowledge_Robotic,
    dtError := Status_GVL.arAlarmActive); // Alarm_Event_Active
HMI_GVL.AlarmOutfeed_Location[34] := AlarmEventHistory[34].bEnable_Out OR AlarmEventActive[34].bEnable_Out;

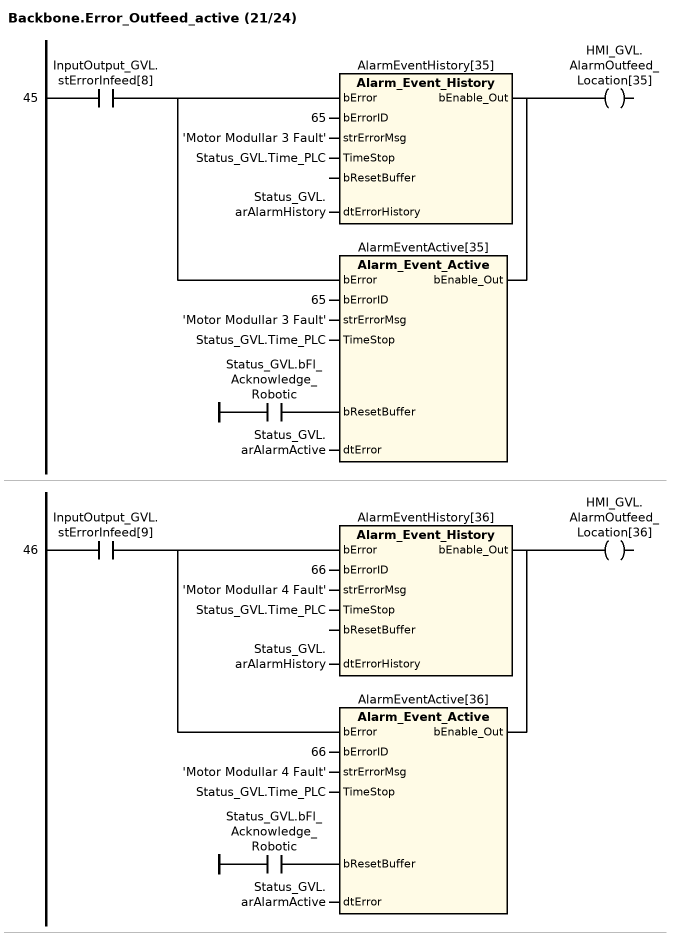
// NETWORK 45
AlarmEventHistory[35](
    bError := InputOutput_GVL.stErrorInfeed[8],
    bErrorID := 65,
    strErrorMsg := 'Motor Modullar 3 Fault',
    TimeStop := Status_GVL.Time_PLC,
    dtErrorHistory := Status_GVL.arAlarmHistory); // Alarm_Event_History
AlarmEventActive[35](
    bError := InputOutput_GVL.stErrorInfeed[8],
    bErrorID := 65,
    strErrorMsg := 'Motor Modullar 3 Fault',
    TimeStop := Status_GVL.Time_PLC,
    bResetBuffer := Status_GVL.bFl_Acknowledge_Robotic,
    dtError := Status_GVL.arAlarmActive); // Alarm_Event_Active
HMI_GVL.AlarmOutfeed_Location[35] := AlarmEventHistory[35].bEnable_Out OR AlarmEventActive[35].bEnable_Out;

// NETWORK 46
AlarmEventHistory[36](
    bError := InputOutput_GVL.stErrorInfeed[9],
    bErrorID := 66,
    strErrorMsg := 'Motor Modullar 4 Fault',
    TimeStop := Status_GVL.Time_PLC,
    dtErrorHistory := Status_GVL.arAlarmHistory); // Alarm_Event_History
AlarmEventActive[36](
    bError := InputOutput_GVL.stErrorInfeed[9],
    bErrorID := 66,
    strErrorMsg := 'Motor Modullar 4 Fault',
    TimeStop := Status_GVL.Time_PLC,
    bResetBuffer := Status_GVL.bFl_Acknowledge_Robotic,
    dtError := Status_GVL.arAlarmActive); // Alarm_Event_Active
HMI_GVL.AlarmOutfeed_Location[36] := AlarmEventHistory[36].bEnable_Out OR AlarmEventActive[36].bEnable_Out;

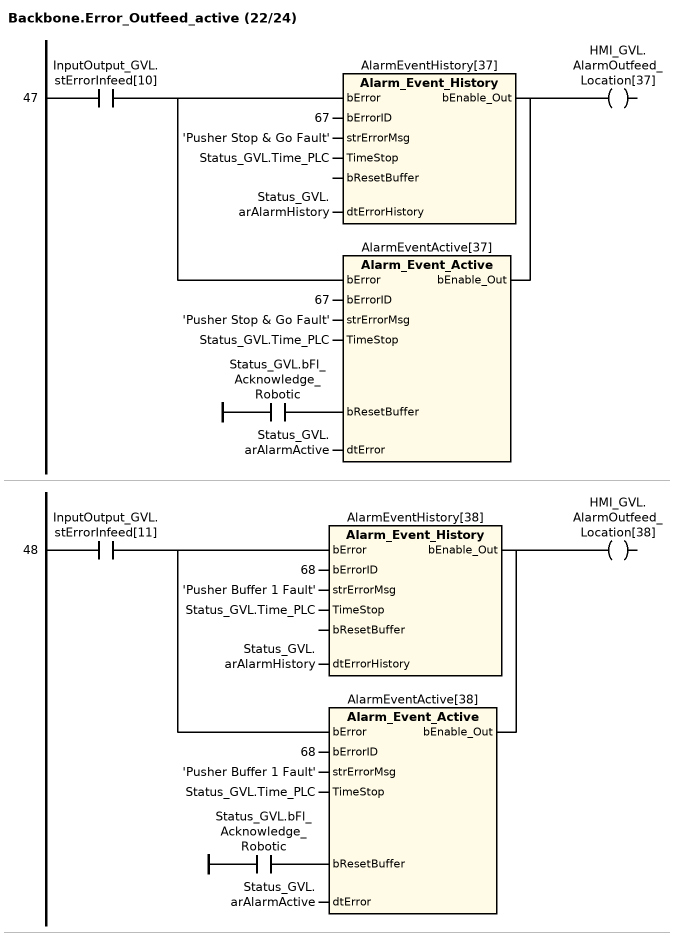
// NETWORK 47
AlarmEventHistory[37](
    bError := InputOutput_GVL.stErrorInfeed[10],
    bErrorID := 67,
    strErrorMsg := 'Pusher Stop & Go Fault',
    TimeStop := Status_GVL.Time_PLC,
    dtErrorHistory := Status_GVL.arAlarmHistory); // Alarm_Event_History
AlarmEventActive[37](
    bError := InputOutput_GVL.stErrorInfeed[10],
    bErrorID := 67,
    strErrorMsg := 'Pusher Stop & Go Fault',
    TimeStop := Status_GVL.Time_PLC,
    bResetBuffer := Status_GVL.bFl_Acknowledge_Robotic,
    dtError := Status_GVL.arAlarmActive); // Alarm_Event_Active
HMI_GVL.AlarmOutfeed_Location[37] := AlarmEventHistory[37].bEnable_Out OR AlarmEventActive[37].bEnable_Out;

// NETWORK 48
AlarmEventHistory[38](
    bError := InputOutput_GVL.stErrorInfeed[11],
    bErrorID := 68,
    strErrorMsg := 'Pusher Buffer 1 Fault',
    TimeStop := Status_GVL.Time_PLC,
    dtErrorHistory := Status_GVL.arAlarmHistory); // Alarm_Event_History
AlarmEventActive[38](
    bError := InputOutput_GVL.stErrorInfeed[11],
    bErrorID := 68,
    strErrorMsg := 'Pusher Buffer 1 Fault',
    TimeStop := Status_GVL.Time_PLC,
    bResetBuffer := Status_GVL.bFl_Acknowledge_Robotic,
    dtError := Status_GVL.arAlarmActive); // Alarm_Event_Active
HMI_GVL.AlarmOutfeed_Location[38] := AlarmEventHistory[38].bEnable_Out OR AlarmEventActive[38].bEnable_Out;

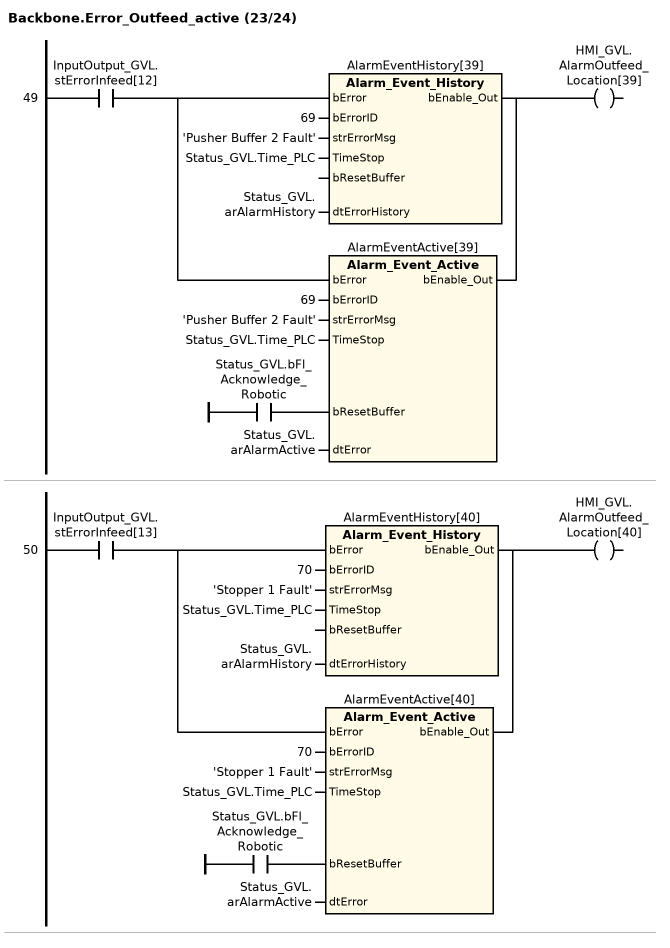
// NETWORK 49
AlarmEventHistory[39](
    bError := InputOutput_GVL.stErrorInfeed[12],
    bErrorID := 69,
    strErrorMsg := 'Pusher Buffer 2 Fault',
    TimeStop := Status_GVL.Time_PLC,
    dtErrorHistory := Status_GVL.arAlarmHistory); // Alarm_Event_History
AlarmEventActive[39](
    bError := InputOutput_GVL.stErrorInfeed[12],
    bErrorID := 69,
    strErrorMsg := 'Pusher Buffer 2 Fault',
    TimeStop := Status_GVL.Time_PLC,
    bResetBuffer := Status_GVL.bFl_Acknowledge_Robotic,
    dtError := Status_GVL.arAlarmActive); // Alarm_Event_Active
HMI_GVL.AlarmOutfeed_Location[39] := AlarmEventHistory[39].bEnable_Out OR AlarmEventActive[39].bEnable_Out;

// NETWORK 50
AlarmEventHistory[40](
    bError := InputOutput_GVL.stErrorInfeed[13],
    bErrorID := 70,
    strErrorMsg := 'Stopper 1 Fault',
    TimeStop := Status_GVL.Time_PLC,
    dtErrorHistory := Status_GVL.arAlarmHistory); // Alarm_Event_History
AlarmEventActive[40](
    bError := InputOutput_GVL.stErrorInfeed[13],
    bErrorID := 70,
    strErrorMsg := 'Stopper 1 Fault',
    TimeStop := Status_GVL.Time_PLC,
    bResetBuffer := Status_GVL.bFl_Acknowledge_Robotic,
    dtError := Status_GVL.arAlarmActive); // Alarm_Event_Active
HMI_GVL.AlarmOutfeed_Location[40] := AlarmEventHistory[40].bEnable_Out OR AlarmEventActive[40].bEnable_Out;

